Staubli VAL3: _globals.pgx

program _globals()
begin
    //\brief
  //
  //\version
  //4.3c
  //
//!version 4.3c
end
